{attribute 'qualified_only'}
VAR_GLOBAL
	bRunning : BOOL;
	bManual : BOOL;
	bAuto : BOOL;
END_VAR

(* stored: Version 1.1.0.1, ProductVersion 3.1.4024.12
   GVL G_Mode: Id {a89507da-b50b-4379-9e9a-399fcb20c7fd} *)
